FUNCTION proj0_TupleStruct_1: DINT
VAR_INPUT
    tuple: TupleStruct_1;
END_VAR

proj0_TupleStruct_1 := tuple.field0;

END_FUNCTION

(* stored: ProductVersion 3.1.0.18, Version 1.1.0.1 *)
